// TIA Portal project "Random with LGF" (V17)

(* hardware
DEVICE "S7-1200 station_1"  S7-1200 Station
   slot 0: "Rack_0"  S7-1200 Rack  Rack  V1.0
   slot 1: "Random Number with Cyclic Interrupt"  CPU 1214C DC/DC/DC  6ES7 214-1AG40-0XB0  V4.5
*)

// ===== PLC "Random Number with Cyclic Interrupt"  CPU 1214C DC/DC/DC =====

VAR_GLOBAL   // PLC tag table "Default tag table"
   "Blue_Light" AT %Q0.0 : Bool;
   "Stop button (NC)" AT %I0.0 : Bool;
   "Red_Light" AT %Q0.4 : Bool;
   "Yellow_Light" AT %Q0.5 : Bool;
   "Green_Light" AT %Q0.6 : Bool;
   "White_Light" AT %Q0.7 : Bool;
   "AlwaysTRUE" AT %M1.2 : Bool;
   "AlwaysFALSE" AT %M1.3 : Bool;
   "Clock_Byte" AT %MB0 : Byte;
   "Clock_10Hz" AT %M0.0 : Bool;
   "Clock_5Hz" AT %M0.1 : Bool;
   "Clock_2.5Hz" AT %M0.2 : Bool;
   "Clock_2Hz" AT %M0.3 : Bool;
   "Clock_1.25Hz" AT %M0.4 : Bool;
   "Clock_1Hz" AT %M0.5 : Bool;
   "Clock_0.625Hz" AT %M0.6 : Bool;
   "Clock_0.5Hz" AT %M0.7 : Bool;
   "Reset_up" AT %M2.1 : Bool;
   "System_Byte" AT %MB1 : Byte;
   "Start Button" AT %I0.1 : Bool;
   "Running" AT %M3.2 : Bool;
   "RNG_done" AT %M3.3 : Bool;
   "Enable_Random_Out" AT %M3.4 : Bool;
   "Starting" AT %M1.0 : Bool;
   "Start_done" AT %M3.1 : Bool;
END_VAR

DATA_BLOCK "RND# Generator DB"   // DB1
{ S7_Optimized_Access := 'TRUE' }
VERSION : 0.1
   VAR
      min_rand : Word := 0;
      max_rand : Word := 100;
      random_val : Word;
      error : Bool;
      status : Word;
      sub_status : Word;
   END_VAR
BEGIN
END_DATA_BLOCK

ORGANIZATION_BLOCK "Main"   // OB1, LAD, ProgramCycle
TITLE = "Main Program Sweep (Cycle)"
{ S7_Optimized_Access := 'TRUE' }
VERSION : 0.1
// Author: Andi Sama
// Organization: Sinergi Wahana Gemilang
// Date (created): Jan 19, 2023
// Date (last modified): Jan 20, 2023
// 
// Purpose: Experimeting with Library of Generic Functions: Random Number Generator
// - Real PLC: Siemens PLC 1200 DC/DC/DC
// 
// Program Logic
// 
// Execute [OB100]
// # in Main [OB1]
// DO
//   If Start_Push_Button  is Pressed
//      Energize Blue_LED with 2Hz frequency
//       #Generate random number every 250 mS  by interrupt
//      With Cyclic_Interrupt (every 250 mS)
//        random_val="RND# Generator" [OB30] with min=0, max=100  
//      Energize Red_Light if 0<=random_val<=25
//      Energize Yellow_Light if 25<=random_val<=50
//      Energize Yellow_Light if 50<=random_val<=75
//      Energize Yellow_Light if 75<=random_val<=100
//   End
// UNTIL Stop_Push_Button is Pressed
   VAR_INPUT
      Initial_Call : Bool;   // Initial call of this OB
      Remanence : Bool;   // =True, if remanent data are available
   END_VAR
   VAR_TEMP
      Start : Bool;
      Start_done : Bool;
      PLC_Initialized : Bool;
      CounterValue : Int;
   END_VAR
   VAR CONSTANT
      Input_Lowest : Word := 0;
      Input_Low : Word := 25;
      Input_Mid : Word := 50;
      Input_High : Word := 75;
      Input_Highest : Word := 100;
      PLC_ADC_Max : Int := 5;
   END_VAR
   VAR_TEMP   // added for the SCL form of the ladder/FBD networks
      _w1 : Bool;
   END_VAR
BEGIN

REGION Network 1: Preparation
   // Real PLC
   // - Directly gets analog input (0-10VDC or 4-20mA) from PLC Analog Input (CH00)
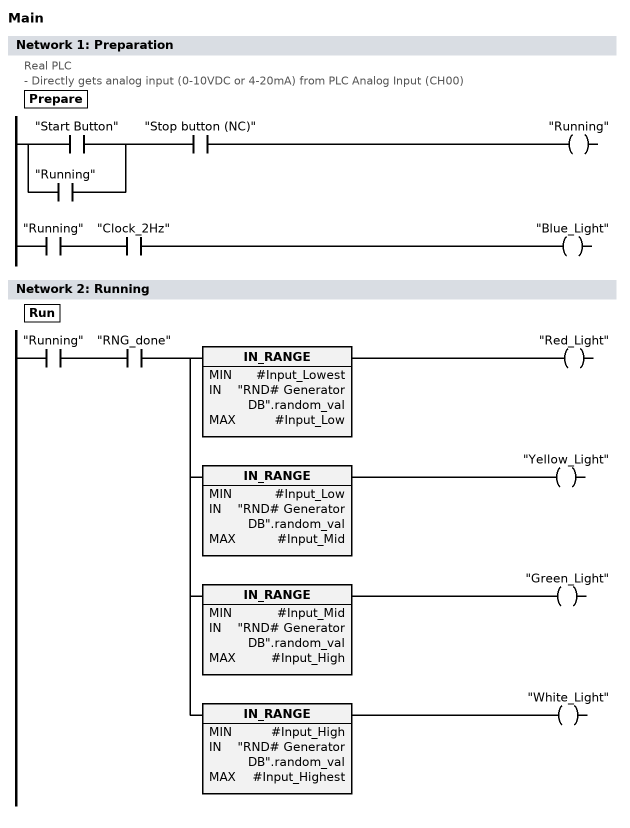
   Label( Prepare )
   RUNG wire#powerrail
      Contact( "Start Button" )
      wire#w1
      Contact( "Stop button (NC)" )
      Coil( "Running" )
   END_RUNG
   RUNG wire#powerrail
      Contact( "Running" )
   END_RUNG wire#w1
   RUNG wire#powerrail
      Contact( "Running" )
      Contact( "Clock_2Hz" )
      Coil( "Blue_Light" )
   END_RUNG
   // the same network as SCL:
   Prepare:
   "Running" := ("Start Button" OR "Running") AND "Stop button (NC)";
   "Blue_Light" := "Running" AND "Clock_2Hz";
END_REGION

REGION Network 2: Running
   Label( Run )
   RUNG wire#powerrail
      Contact( "Running" )
      Contact( "RNG_done" )
      wire#w1
      { S7_Templates := "SrcType := DInt" } InRange(min := #Input_Lowest, in := "RND# Generator DB".random_val, max := #Input_Low)
      Coil( "Red_Light" )
   END_RUNG
   RUNG wire#w1
      { S7_Templates := "SrcType := DInt" } InRange(min := #Input_Low, in := "RND# Generator DB".random_val, max := #Input_Mid)
      Coil( "Yellow_Light" )
   END_RUNG
   RUNG wire#w1
      { S7_Templates := "SrcType := DInt" } InRange(min := #Input_Mid, in := "RND# Generator DB".random_val, max := #Input_High)
      Coil( "Green_Light" )
   END_RUNG
   RUNG wire#w1
      { S7_Templates := "SrcType := DInt" } InRange(min := #Input_High, in := "RND# Generator DB".random_val, max := #Input_Highest)
      Coil( "White_Light" )
   END_RUNG
   // the same network as SCL:
   Run:
   #_w1 := "Running" AND "RNG_done";
   "Red_Light" := #_w1 AND (#Input_Lowest <= "RND# Generator DB".random_val) AND ("RND# Generator DB".random_val <= #Input_Low);
   "Yellow_Light" := #_w1 AND (#Input_Low <= "RND# Generator DB".random_val) AND ("RND# Generator DB".random_val <= #Input_Mid);
   "Green_Light" := #_w1 AND (#Input_Mid <= "RND# Generator DB".random_val) AND ("RND# Generator DB".random_val <= #Input_High);
   "White_Light" := #_w1 AND (#Input_High <= "RND# Generator DB".random_val) AND ("RND# Generator DB".random_val <= #Input_Highest);
END_REGION
END_ORGANIZATION_BLOCK

ORGANIZATION_BLOCK "RND# Generator"   // OB30, LAD, CyclicInterrupt
{ S7_Optimized_Access := 'TRUE' }
VERSION : 0.1
   VAR_INPUT
      Initial_Call : Bool;   // Initial call of this OB
      Event_Count : Int;   // Events discarded
   END_VAR
   VAR_TEMP   // added for the SCL form of the ladder/FBD networks
      _w1 : Bool;
   END_VAR
BEGIN

REGION Network 1
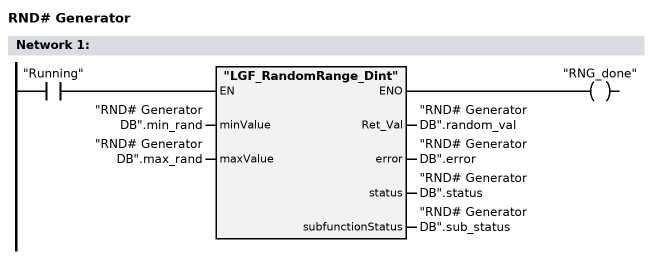
   RUNG wire#powerrail
      Contact( "Running" )
      "LGF_RandomRange_Dint"(minValue := "RND# Generator DB".min_rand, maxValue := "RND# Generator DB".max_rand, Ret_Val => "RND# Generator DB".random_val, error => "RND# Generator DB".error, status => "RND# Generator DB".status, subfunctionStatus => "RND# Generator DB".sub_status)
      Coil( "RNG_done" )
   END_RUNG
   // the same network as SCL:
   "RND# Generator DB".random_val := "LGF_RandomRange_Dint"(EN := "Running",
                           minValue := "RND# Generator DB".min_rand,
                           maxValue := "RND# Generator DB".max_rand,
                           error => "RND# Generator DB".error,
                           status => "RND# Generator DB".status,
                           subfunctionStatus => "RND# Generator DB".sub_status,
                           ENO => #_w1);
   "RNG_done" := #_w1;
END_REGION
END_ORGANIZATION_BLOCK

ORGANIZATION_BLOCK "Initialization"   // OB100, LAD, Startup
TITLE = "Complete Restart"
{ S7_Optimized_Access := 'TRUE' }
VERSION : 0.1
   VAR_INPUT
      LostRetentive : Bool;   // True if retentive data are lost
      LostRTC : Bool;   // True if date and time are lost
   END_VAR
BEGIN

REGION Network 1: Start
   // Select one of Run Modes:
   // 1: Real PLC 
   // 2: PLC Simulator
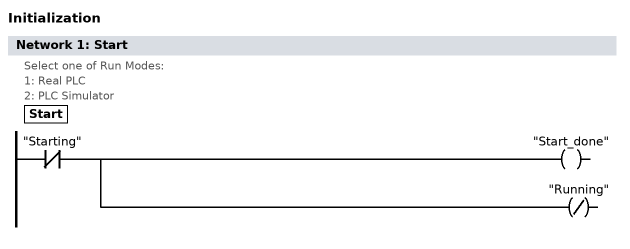
   Label( Start )
   RUNG wire#powerrail
      I_Contact( "Starting" )
      wire#w1
      Coil( "Start_done" )
   END_RUNG
   RUNG wire#w1
      I_Coil( "Running" )
   END_RUNG
   // the same network as SCL:
   Start:
   "Start_done" := NOT "Starting";
   "Running" := NOT (NOT "Starting");
END_REGION
END_ORGANIZATION_BLOCK

// folder: LGF/4 Math operations

FUNCTION "LGF_RandomRange_Dint" : DInt   // FC10013, SCL
TITLE = LGF_RandomRange_DInt
{ S7_Optimized_Access := 'TRUE' }
AUTHOR : Siemens_Digital_Industries
FAMILY : LGF
NAME : LGF_RandomRange_DInt
// This function generates a random value in defined limits with each call.  
// The random number has the data type DInt in the specified range.
// Diese Funktion generiert bei jedem Aufruf einen zufälligen Wert zwischen einem definierten Max- und Minwert.  
// Die Zufallszahl hat den Datentyp DInt im spezifiziertem Wertebereich.
   VAR_INPUT
      minValue : DInt;   // Minimalwert der für den Wertebereich der Zufallszahl - Untergrenze / Minimum value of the range of the random number - lower border
      maxValue : DInt;   // Maximalwert der für den Wertebereich der Zufallszahl - Obergrenze / Maximum value of the range of the random number - upper border
   END_VAR
   VAR_OUTPUT
      error : Bool;   // FALSE: No error TRUE: An error occurred during the execution of the FB / FALSE: Kein Fehler TRUE: Während der Ausführung des FB ist ein Fehler aufgetreten
      status : Word;   // 16#0000-16#7FFF: Status of the FB 16#8000-16#FFFF: Error identification (see following Table) / 16#0000-16#7FFF: Status des FB 16#8000-16#FFFF: Fehleridentifikation (siehe folgende Tabelle)
      subfunctionStatus : Word;   // Status or return value of called FB's, FC's and system blocks / Status oder Rückgabewert von aufgerufenen FB's / FC's und Systemfunktionen
   END_VAR
   VAR_TEMP
      tempTime : DTL;   // Temp memory for System time / Temp variable für System Zeit
      tempNanoSecondInDWord : DWord;   // Temp UDInt converted to DWord for access to individual bytes / Temp UDInt konvertiert nach Dword für den Zufriff per Slice auf die Bytes
      tempTimeStatus : Word;   // Temp status of the instruction `RD_SYS_T` / Temp Status der Systemfunktion `RD_SYS_T`
      tempRandomValue : DWord;   // Temp Random startvalue / Temp Zufallswert als Startwert
      tempNormReal : Real;   // Temp normalized Real value (0.0 - 1.0) / Temp Normalisierer Realwert (0.0 - 1.0)
   END_VAR
   // Ret_Val : Random Real number in the predefined range / Zufallszahl vom Datentyp Real im definierten Wertebereich
   VAR CONSTANT
      ZERO : DInt := 0;   // Zero / 0.0 - value in case of error / Null / 0.0 - Rückgabewert im Fehlerfall
      MAX_UDINT : UDInt := 4294967295 ;   // Maximum DInt datatype / Maximalwert eines DInt Datentype
      SUB_STATUS_NO_ERROR : Word := 16#0000;   // Status: sub function call ends without error / Status: Unterfunktionsaufruf ohne Fehler beendet
      STATUS_FINISHED_NO_ERROR : Word := 16#0000;   // Execution finished without errors / Abarbeitung ohne Fehler beendet
      ERR_MAX_LESS_MIN : Word := 16#8200;   // Error: The ranges specified are wrong: `minValue` is greater than `maxValue` / Fehler: Der spezifizierte Wetebereich is fehlerhaft: `minValue` ist größer als `maxValue`
      ERR_RD_SYS_T : Word := 16#8600;   // Error in `RD_SYS_T` command - check `subFunctionStatus` code / Fehler in Anweisung `RD_SYS_T` - weitere infos in `subFunctionStatus`
   END_VAR
BEGIN
   REGION Block info header
     //=============================================================================
     // SIEMENS AG / (c)Copyright 2017
     //-----------------------------------------------------------------------------
     // Title:            LGF_RandomRange_DInt
     // Comment/Function: This function generates random numbers in defined limits (Datatype DInt)
     // Library/Family:   LGF(Library General Functions)
     // Author:           Siemens Digital Industry Support
     // Tested with:      S7-PLCSIM Advanced V2.0 SP1
     // Engineering:      TIA Portal V15 Update 2
     // Restrictions:     ENO disabled - error handling done by error and status
     // Requirements:     PLC (S7-1200 / S7-1500)
     //-------------------------------------------------------------------------------
     // Change log table:
     // Version  | Date       | Expert in charge       | Changes applied
     //----------|------------|------------------------|------------------------------
     // 01.00.00 19.08.2015  Siemens Industry Online Support
     //                      First released version
     // 01.00.01 02.01.2017  Siemens Industry Online Support
     //                      Upgrade: TIA Portal V14 Update 1
     // 01.00.02 17.08.2018  Siemens Industry Online Support
     //                      Upgrade: TIA V15 Update 2
     // 01.00.03 23.11.2018  Siemens Industry Online Support
     //                      Upgrade: TIA V15.1
     // 01.01.00 09.10.2019  Simatic Systems Support
     //                      Renamed from "LGF_RandomInt" to "LGF_RandomRange_DInt"
     //                      change random datatype from Int to DInt
     //                      Regions, comments and constants are added
     // 03.00.00 23.04.2020  Simatic Systems Support
     //                      Set version to V3.0.0, harmonize the version of the whole library
     // 03.00.01 04.02.2021  Simatic Systems Support
     //                      Insert documentation
     //=============================================================================
   END_REGION Block info header

   REGION DESCRIPTION
     (/*Note
   :    The status of called commands is output in `subFunctionStatus`. In this case, the output value in `status` indicates which command caused the error. In this case, refer to the TIA Portal Online Help section for information on the respective commands.

   The block generates random values that are between the specified `minValue` and the `maxValue`. This random value is output via the `Ret_Val`.

   The random value is formed from the nanoseconds of the current system time of the CPU. The byte order of this value is inverted and then converted to a DInt.
   Hinweis
   :    In `subFunctionStatus` wird der Status von aufgerufenen Anweisungen ausgegeben. Der Ausgangswert in `status` gibt in diesem Fall an, welche Anweisung den Fehler verursacht hat. Holen Sie sich in diesem Fall die Informationen aus der TIA Portal Online Hilfe zu den jeweiligen Anweisungen.

   Der Baustein generiert zufällige Werte, die zwischen dem angegebenen `minValue`-Wert und `maxValue`-Wert liegen. Dieser zufällige Wert wird über den `Ret_Val` ausgegeben.

   Der Zufallswert wird aus den Nanosekunden der aktuellen Systemzeit der CPU gebildet. Dabei wird die Bytereihenfolge dieses Wertes invertiert und anschließend in eine DInt ungewandelt.*/)
   END_REGION DESCRIPTION

   REGION Validation
     // Check if the maximal Value is less than the minimal value
     IF (#minValue > #maxValue) THEN
       #error := true;
       #status := #ERR_MAX_LESS_MIN;
       #subfunctionStatus := #SUB_STATUS_NO_ERROR;
       #LGF_RandomRange_Dint := #ZERO;
       RETURN;
     END_IF;

     // Read system time
     #tempTimeStatus := INT_TO_WORD(RD_SYS_T(#tempTime));

     // Check return variable for error
     IF (#tempTimeStatus <> #SUB_STATUS_NO_ERROR) THEN
       #error := true;
       #status := #ERR_RD_SYS_T;
       #subfunctionStatus := #tempTimeStatus;
       #LGF_RandomRange_Dint := #ZERO;
       RETURN;
     END_IF;
   END_REGION

   REGION Calculating random number
     // Converting to double word so individual bytes can be addressed
     #tempNanoSecondInDWord := UDINT_TO_DWORD(#tempTime.NANOSECOND);

     // Callculate a random-start-value depending on the time
     #tempRandomValue.%B3 := #tempNanoSecondInDWord.%B0;
     #tempRandomValue.%B2 := #tempNanoSecondInDWord.%B1;
     #tempRandomValue.%B1 := #tempNanoSecondInDWord.%B2;
     #tempRandomValue.%B0 := #tempNanoSecondInDWord.%B3;

     // Norm the calculated random number: 0.0 <= #tempNormReal <= 1.0
     #tempNormReal := UDINT_TO_REAL(DWORD_TO_UDINT(#tempRandomValue)) / UDINT_TO_REAL(#MAX_UDINT);

     // Scale the tempNormReal to be in the range of maxValue and minValue
     #LGF_RandomRange_Dint := REAL_TO_DINT((#tempNormReal * DINT_TO_REAL(#maxValue - #minValue) + DINT_TO_REAL(#minValue)));

     #error := false;
     #status := #STATUS_FINISHED_NO_ERROR;
     #subfunctionStatus := #SUB_STATUS_NO_ERROR;
     // ENO mechanism is not used
     ENO := TRUE;
   END_REGION
END_FUNCTION